KUKA KRL data list: InitializationModule.dat

&ACCESS RV
DEFDAT InitializationModule PUBLIC

   ;WAYPOINTS

ENDDAT
